FUNCTION_BLOCK FB_SimFiller
VAR_INPUT
END_VAR
VAR_OUTPUT
END_VAR
VAR
	fVolumeFilled				AT %Q* : LREAL;
	bFillValve					AT %I* : BOOL;
	bPartPresent				AT %Q* : BOOL;
	
	rand						: DRAND;
	iState						: DINT;
END_VAR
VAR CONSTANT
	FLOW_RATE					: LREAL := 1.0;
END_VAR

rand(Seed:=113);

CASE iState OF
	0:
		IF bFillValve THEN
			iState := 10;
		ELSE
			fVolumeFilled := 0.0;
		END_IF
		
	10:
		IF bFillValve THEN
			fVolumeFilled := fVolumeFilled + (FLOW_RATE + rand.Num);
		ELSE
			iState := 20;
		END_IF
		
	20:
		iState := 0;
		
END_CASE

END_FUNCTION_BLOCK

(* stored: Version 1.1.0.1, ProductVersion 3.1.4024.12
   POU FB_SimFiller: Id {45f26f00-5e10-4615-86cf-ae8ecf9db752}, SpecialFunc None *)
